PROGRAM CogenerationProcess
VAR

(**************MIXIT obiegi grzewcze*******************************************)	
	fbMixit_C01		: FB_Mixit; //Mixit MX01 obiegu chłodnicy kogeneratora C01 - regulacja chłodzenia
	fbMixit_R01		: FB_Mixit; //Mixit MX02 obiegu podgrzewania reaktora R01 - regulacja ogrzewanie
	fbMixit_EX01	: FB_Mixit; //Mixit MX03 obiegu podgrzewania wymiennika osuszacza EX-01 - podgrzewanie ciągłe
	fbMixit_H01	    : FB_Mixit; //Mixit MX04 obiegu nagrzewnicy H0-1 - regulacja ogrzewania

(************** Temp Sensory **************************************************)
	fbTempSens_HC01	: FB_Scaling; //Czujnik temperatury w sprzegle hydffraulicznym HC01	
	fbMedian5       : FB_Median5;	//filtr medianowy do czujnika temperatury
	
(************** DACHS CONTROL *************************************************)
	fbDachsControl  : FB_DachsControl;	
	
	
END_VAR

ACT_TempSens(); //skalowanie i zapisywanie do GVL z czujników temperatury
ACT_DachsControl();


//obsługa obiegu chłodnicy C01 z regulacja dwustawnowa  jesli temperatura za wysoka to wlacz chlodnice jesli nie wylacz 
fbMixit_C01.MixitCv(Sensor := GVL_Cogeneration.TempSens_HC01); //pobierz i ustaw temperature aktualna np z bloku skalowania temperatury
fbMixit_C01.MixitState(IO := GVL_Cogeneration.stMixit_C01); // pobiera dostep do struktury poprzez VAR_IN_OUT i wykonuje program 

//obsługa obiegu reaktora R01 z regulacją dwustawnową temperatry
fbMixit_R01.MixitCv(Sensor := GVL_Fermentation.TempSens_R01);
fbMixit_R01.MixitState(IO := GVL_Cogeneration.stMixit_R01); // pobiera dostep do struktury poprzez VAR_IN_OUT i wykonuje program 

//obsługa obiegu podgrzewacza EX01 bez regulacji
fbMixit_EX01.MixitState(IO := GVL_Cogeneration.stMixit_EX01); // pobiera dostep do struktury poprzez VAR_IN_OUT i wykonuje program 

//obsługa obiegu nagrzewnicy hali H01 bez regulacji
fbMixit_H01.MixitCv(Sensor := GVL_Fertilizer.TempSens_H01);
fbMixit_H01.MixitState(IO := GVL_Cogeneration.stMixit_H01); // pobiera dostep do struktury poprzez VAR_IN_OUT i wykonuje program

ACTION ACT_DachsControl:
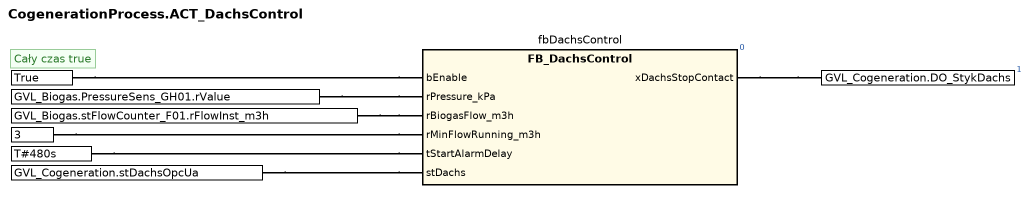
// Cały czas true
fbDachsControl(
    bEnable := True,
    rPressure_kPa := GVL_Biogas.PressureSens_GH01.rValue,
    rBiogasFlow_m3h := GVL_Biogas.stFlowCounter_F01.rFlowInst_m3h,
    rMinFlowRunning_m3h := 3,
    tStartAlarmDelay := T#480s,
    stDachs := GVL_Cogeneration.stDachsOpcUa); // FB_DachsControl
GVL_Cogeneration.DO_StykDachs := fbDachsControl.xDachsStopContact;
END_ACTION

ACTION ACT_TempSens:
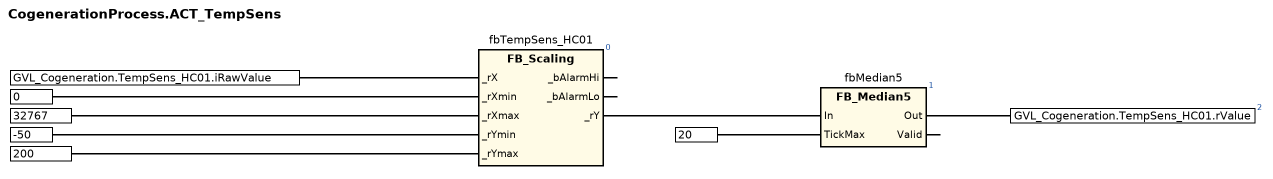
fbTempSens_HC01(
    _rX := GVL_Cogeneration.TempSens_HC01.iRawValue,
    _rXmin := 0,
    _rXmax := 32767,
    _rYmin := -50,
    _rYmax := 200); // FB_Scaling
fbMedian5(In := fbTempSens_HC01._rY, TickMax := 20); // FB_Median5
GVL_Cogeneration.TempSens_HC01.rValue := fbMedian5.Out;
END_ACTION

END_PROGRAM

(* stored: Version 1.1.0.1, ProductVersion 3.1.4024.16
   POU CogenerationProcess: Id {40f1c5ca-73b7-47a7-b437-7b9b210b8155}, SpecialFunc None
   Action ACT_DachsControl: Id {5be6a338-00de-4dcb-bc01-8d305d5d5d21}
   Action ACT_TempSens: Id {69d8c34b-c1cd-4ec1-9c8f-33fba772cae6} *)
